Staubli VAL3: buildListFrame.pgx

program buildListFrame(num x_nIndex)
  local num l_nSize
  local string l_sEvent
  local num i
  local string l_sEmpty
  local string l_sItem
begin
  // Build the list
  call use:setSizeList(15,0,15,11)
  call use:listcreate("FRAME")
  // insert all the element
  for i=0 to size(saveData:fFrameItem)-1
    l_sItem=toString("2",i)+" "+saveData:fFrameItem[i].sName
    call use:listadd(l_sItem)
  endFor
  // update it
  call use:listupdate(0)
  call use:selectNewField(x_nIndex,x_nIndex,x_nIndex)
  // leave ...
end
